(* IEC 61131-3 sources: ICSML/Codesys_V3/Function Blocks/Sequential.pou, 1 file *)

(* ---- Sequential.pou ---- *)
(*#-#-#-#-#-#-#-#-#-#---Declaration---#-#-#-#-#-#-#-#-#-#-#-#-#*)

FUNCTION_BLOCK Sequential IMPLEMENTS Model
VAR
	layers_i: POINTER TO Layer;
	layers_num_i: INT;
END_VAR

(*#-#-#-#-#-#-#-#-#-#---Implementation---#-#-#-#-#-#-#-#-#-#-#-#-#*)
